Staubli VAL3: Day8.pjx

--- Day8.pjx ---
Parameters version=s8.13.1Cs9_BS2800 stackSize=5000 millimeterUnit=true
Program file=start.pgx
Program file=stop.pgx
Data file=Day8.dtx
Library alias=util path=Disk://helpers/helpers.pjx
Library alias=math path=Disk://math/math.pjx
Library alias=str path=Disk://string/string.pjx
Library alias=stat path=Disk://statistics/statistics.pjx
Type name=lists path=Disk://types/lists/lists.pjx

--- Day8.dtx ---
string sInput
lists lResult
  [0]
    string sString
lists lResultSplit
  [0]
    string sString

--- start.pgx ---
program start()
  local num l_nElement
  local num l_nString
  local num l_nResult
begin

  // read file
  call util:readFile("Disk://input_day8.txt", sInput)
  // sInput[0] = "begfcd fabg aecgbdf ..... | cbgef befdcg bceaf fagb"

  call str:splitString(sInput," | ", lResult)
  // lResult.sString[0] = "begfcd fabg aecgbdf ...."
  // lResult.sString[1] = "cbgef befdcg bceaf fagb"

  // PUZZLE 1
  l_nResult = 0
  for l_nElement = 0 to size(lResult)-1
    call str:splitString(lResult[l_nElement].sString[1], " ", lResultSplit)
    for l_nString = 0 to size(lResultSplit.sString)-1
      // check if stringlength is 2 (#1), 3 (#7), 4 (#4) or 7 (#8)
      if len(lResultSplit.sString[l_nString]) == 2 or len(lResultSplit.sString[l_nString]) ==3 or len(lResultSplit.sString[l_nString]) == 4 or len(lResultSplit.sString[l_nString]) == 7
        l_nResult = l_nResult+1
      endIf
    endFor
  endFor

  call util:printNum(l_nResult)
  // 367

end
